(* CoDeSys 2.3 library: BusDiag.lib *)

(* POU DiagGetBusState, ST *)
FUNCTION_BLOCK DiagGetBusState
VAR_INPUT
	ENABLE:BOOL ;
	DRIVERNAME:POINTER TO STRING ;
	DEVICENUMBER:INT ;
END_VAR
VAR_OUTPUT
	READY: BOOL ;
	STATE:INT ;
	EXTENDEDINFO:ARRAY[0..129] OF BYTE ;
END_VAR
VAR
	BOLDENABLE:BOOL ;
END_VAR
;
END_FUNCTION_BLOCK

(* POU DiagGetState, ST *)
FUNCTION_BLOCK DiagGetState
VAR_INPUT
	ENABLE:BOOL ;
	DRIVERNAME:POINTER TO STRING ;
	DEVICENUMBER:INT ;
	BUSMEMBERID:DWORD ;
END_VAR
VAR_OUTPUT
	READY: BOOL ;
	STATE:INT ;
	EXTENDEDINFO:ARRAY[0..99] OF BYTE ;
END_VAR
VAR
	BOLDENABLE:BOOL ;
END_VAR
;
END_FUNCTION_BLOCK

(* POU DiagSetBusState, ST *)
FUNCTION_BLOCK DiagSetBusState
VAR_INPUT
	ENABLE:BOOL ;
	DRIVERNAME:POINTER TO STRING ;
	DEVICENUMBER:INT ;
	NEWSTATE:INT ;
END_VAR
VAR_OUTPUT
	READY: BOOL ;
	STATE:INT ;
END_VAR
VAR
	BOLDENABLE:BOOL ;
END_VAR
;
END_FUNCTION_BLOCK

(* POU DiagSetState, ST *)
FUNCTION_BLOCK DiagSetState
VAR_INPUT
	ENABLE:BOOL ;
	DRIVERNAME:POINTER TO STRING ;
	DEVICENUMBER:INT ;
	NEWSTATE:INT ;
	BUSMEMBERID:DWORD ;
END_VAR
VAR_OUTPUT
	READY: BOOL ;
	STATE:INT ;
END_VAR
VAR
	BOLDENABLE:BOOL ;
END_VAR
;
END_FUNCTION_BLOCK
